(* IEC 61131-3 sources: Fosela-House-/control/free_evolution, 19 files *)

(* ---- GVL_Evolution.st ---- *)
(* ============================================================
   GVL_Evolution.st
   Variables globales del controlador principal (maestro Modbus).
   Sistema principal — Fosela House
   Arquitectura: BC monobloc genérica (sin HTR) + solar térmico
   ============================================================ *)

VAR_GLOBAL

    (* ---- Entradas analógicas locales (TT4-TT13) ---- *)
    TT4             : REAL;     (* D1 fondo — retorno agua técnica fría [°C] *)
    TT5             : REAL;     (* D2 cabeza — agua técnica caliente, salida a consumos [°C] *)
    TT6             : REAL;     (* Buffer D3 cabeza [°C] *)
    TT7             : REAL;     (* Buffer D3 fondo [°C] *)
    TT8             : REAL;     (* Ida primario BC [°C] *)
    TT9             : REAL;     (* Retorno primario BC [°C] *)
    TT11            : REAL;     (* Temperatura piscina [°C] *)
    TT12            : REAL;     (* Exterior [°C] *)
    TT13            : REAL;     (* Retorno fancoils [°C] *)

    (* ---- Entradas digitales ---- *)
    DI_Z1           : BOOL;     (* Termostato seguridad D1 activo *)
    DI_Z2           : BOOL;     (* Termostato seguridad D2 activo *)
    DI_INUND_FC     : BOOL;     (* Sensor inundación bandejas fancoils *)
    DI_BDC_FAULT    : BOOL;     (* Fallo BC (señal de la propia unidad) *)
    DI_IF_PISC      : BOOL;     (* Interruptor de flujo piscina *)

    (* ---- Salidas digitales ---- *)
    (* Distribución producción BC — dos V3V en cascada:
       V3V1: FALSE=Reservorio (D2 serpentines)  TRUE=→V3V2
       V3V2: FALSE=Buffer D3 fancoils           TRUE=HX_BC piscina *)
    DO_V3V1         : BOOL;     (* BC primario: FALSE=reservorio, TRUE=no-reservorio *)
    DO_V3V2         : BOOL;     (* no-reservorio: FALSE=fancoils (D3), TRUE=piscina (HX_BC) *)
    DO_VP_HX_SOLAR  : BOOL;     (* Válvula piscina lado HX solar *)
    DO_VP_HX_BC     : BOOL;     (* Válvula piscina lado HX aerotérmico *)
    DO_V3V_APT_01   : BOOL;     (* Aparto 1: FALSE=agua precalentada, TRUE=AFS red *)
    DO_V3V_APT_02   : BOOL;
    DO_V3V_APT_03   : BOOL;
    DO_V3V_APT_04   : BOOL;
    DO_P3           : BOOL;     (* Bomba fancoils arranque *)

    (* ---- Datos recibidos del controlador solar por Modbus ---- *)
    SM              : ST_SolarData;  (* Ver Types_Common.st *)

    (* ---- Modos y estados del sistema ---- *)
    bdc_mode        : E_BDC_Mode   := BDC_OFF;
    bdc_priority    : E_BDC_Priority := PRIO_ACS_CLIMATE_POOL;
    bc_mode_heat    : BOOL := TRUE;   (* TRUE=calefacción/ACS, FALSE=refrigeración *)

    (* ---- Ciclo de pasteurización ---- *)
    hyg_phase      : E_Hygienization_Phase := HYG_IDLE;
    hyg_request    : BOOL := FALSE;
    hyg_apt_idx    : UINT := 1;

    (* ---- Alarmas ---- *)
    alarms          : ST_SystemAlarms;

    (* ---- Setpoints enviados al controlador solar vía Modbus ---- *)
    P10_SolarDeltaTTarget           : UINT := 80;    (* 8.0 K ×10 *)
    P16_MinTempForPoolSolarHeating  : UINT := 750;   (* 75.0°C ×10 *)
    P17_SolarOverheatShutterClose   : UINT := 0;
    P19_SolarMode                   : UINT := 0;
    pool_demand_ext                 : UINT := 0;

END_VAR

(* ---- GVL_HMI_Params.st ---- *)
(* ============================================================
   GVL_HMI_Params.st
   Parámetros editables del HMI con sus rangos y valores por defecto.
   FUENTE ÚNICA DE VERDAD para todos los setpoints del sistema.
   Cualquier modificación desde el panel actualiza estas variables;
   la lógica de control las lee desde aquí.
   ============================================================ *)

VAR_GLOBAL RETAIN  (* RETAIN: sobreviven a un corte de alimentación *)

    (* ---- SOLAR ------------------------------------------ *)
    HMI_SP_DT_solar     : REAL := 8.0;   (* ΔT objetivo P1  [3.0 – 15.0 K]   paso 0.5 *)
    HMI_SP_TT3_pool     : REAL := 75.0;  (* TT3 → piscina   [60.0 – 90.0 °C] paso 1.0 *)
    HMI_modo_solar      : UINT := 0;     (* 0=AUTO 1=ACS 2=PISC 3=OFF *)

    (* ---- ACS -------------------------------------------- *)
    HMI_SP_TT5          : REAL := 65.0;  (* Setpoint D2 cab  [50.0 – 80.0 °C] paso 0.5 *)
    HMI_HS_TT5          : REAL := 3.0;   (* Histéresis TT5   [1.0 – 5.0 K]   paso 0.5 *)
    HMI_SP_TT4_start    : REAL := 50.0;  (* Umbral arrq BDC  [40.0 – 60.0 °C] paso 0.5 *)

    (* ---- CLIMATIZACIÓN ----------------------------------- *)
    HMI_SP_heat         : REAL := 45.0;  (* Setpoint calefac [35.0 – 60.0 °C] paso 0.5 *)
    HMI_SP_cool         : REAL := 9.0;   (* Setpoint refrig  [5.0 – 15.0 °C]  paso 0.5 *)
    HMI_HS_heat         : REAL := 2.0;   (* Histéresis calef [1.0 – 5.0 K]   paso 0.5 *)
    HMI_HS_cool         : REAL := 1.0;   (* Histéresis refrig[0.5 – 3.0 K]   paso 0.5 *)

    (* ---- PISCINA ---------------------------------------- *)
    HMI_SP_pool         : REAL := 27.0;  (* Setpoint piscina [20.0 – 35.0 °C] paso 0.5 *)
    HMI_HS_pool         : REAL := 1.0;   (* Histéresis pisc  [0.5 – 3.0 K]   paso 0.5 *)

    (* ---- PASTEURIZACIÓN --------------------------------- *)
    HMI_SP_past_target  : REAL := 70.0;  (* T objetivo past. [65.0 – 75.0 °C] paso 0.5 *)
    HMI_past_hold_min   : UINT := 60;    (* Tiempo manten.   [30 – 120 min]   paso 5   *)
    HMI_past_flush_min  : UINT := 30;    (* Tiempo purgado   [15 – 60 min]    paso 5   *)

    (* ---- APARTAMENTOS ----------------------------------- *)
    HMI_apt_mode_01     : UINT := 0;     (* 0=PRECALENTADA 1=AFS *)
    HMI_apt_mode_02     : UINT := 0;
    HMI_apt_mode_03     : UINT := 0;
    HMI_apt_mode_04     : UINT := 0;
    HMI_apt_mode_05     : UINT := 0;

    (* ---- CONFIGURACIÓN SISTEMA -------------------------- *)
    HMI_bdc_priority    : UINT := 0;     (* 0=ACS>CLIM>PISC  1=ACS>PISC>CLIM *)
    HMI_mb_slave_addr   : UINT := 1;     (* Dir. Modbus Smart [1 – 247] *)
    HMI_mb_baudrate     : UINT := 1;     (* 0=9600 1=19200 2=38400 *)

    (* ---- PIN DE ACCESO ---------------------------------- *)
    HMI_pin_test        : UINT := 1234;  (* PIN acceso TEST  [0 – 9999] *)
    HMI_pin_cfg         : UINT := 9999;  (* PIN acceso CFG   [0 – 9999] *)

END_VAR

(* ---- Variables de estado HMI (no RETAIN) ---- *)
VAR_GLOBAL

    (* Solicitudes de acción desde panel *)
    HMI_req_past_manual : BOOL := FALSE; (* Pulso: lanzar pasteurización *)
    HMI_req_alm_reset   : BOOL := FALSE; (* Pulso: reset alarmas *)
    HMI_req_factory_rst : BOOL := FALSE; (* Pulso: reset fábrica (CFG) *)

    (* Estado del HMI *)
    HMI_test_active     : BOOL := FALSE; (* Modo test activo *)
    HMI_cfg_active      : BOOL := FALSE; (* Modo config activo *)
    HMI_pin_ok          : BOOL := FALSE; (* PIN validado en sesión *)

    (* Página actual visible *)
    HMI_current_page    : UINT := 0;     (* 0=MAIN 1=SOL 2=ACS … *)

END_VAR

(* ---- FB_ACS.st ---- *)
(* ============================================================
   FB_ACS.st  –  Control de producción de ACS
   BC monobloc genérica (sin HTR).
   La BC puede producir ACS de dos formas según el equipo:
     a) Modo ACS dedicado (BDC_ACS): produce agua caliente 55-65°C
        directamente al reservorio (D2 serpentines).
     b) Inversión de ciclo (ACS como calefacción): misma V3V1,
        igual lógica, la BC produce caliente al reservorio.
   En ambos casos la lógica PLC es idéntica: V3V1 hacia reservorio
   y la BC en el modo que proceda.
   ============================================================ *)
FUNCTION_BLOCK FB_ACS
VAR_INPUT
    TT4             : REAL;  (* D1 fondo — agua técnica fría *)
    TT5             : REAL;  (* D2 cabeza — agua técnica caliente *)
    bdc_available   : BOOL;  (* BC autorizada por árbitro *)
    hyg_active      : BOOL;  (* Ciclo de higienización activo *)
    enabled         : BOOL := TRUE;
END_VAR
VAR_OUTPUT
    cmd_V3V1_reservorio : BOOL;  (* TRUE = BC primario → reservorio (D2) *)
    demand_BDC          : BOOL;  (* Solicitud al árbitro *)
    acs_satisfied       : BOOL;  (* Reservorio en setpoint *)
END_VAR
VAR
    ctrl_TT5    : FB_Hysteresis;
    ctrl_TT4    : FB_Hysteresis;
END_VAR

(* ACS satisfecho cuando TT5 (D2 cabeza) supera la consigna *)
ctrl_TT5(
    measured   := TT5,
    setpoint   := P30_ACSStorageSetPoint,
    hysteresis := P31_ACSStorageHysteresis,
    mode_heat  := TRUE,
    enabled    := enabled
);
acs_satisfied := NOT ctrl_TT5.output;

(* Demanda BC: cuando TT4 (fondo D1) cae bajo el umbral de arranque *)
ctrl_TT4(
    measured   := TT4,
    setpoint   := P32_ACSBDCStartTemp,
    hysteresis := P33_ACSBDCStartHyst,
    mode_heat  := TRUE,
    enabled    := enabled AND NOT acs_satisfied
);
demand_BDC := ctrl_TT4.output OR hyg_active;

(* V3V1: BC primario hacia reservorio cuando está autorizado *)
cmd_V3V1_reservorio := bdc_available AND (demand_BDC OR hyg_active);

END_FUNCTION_BLOCK

(* ---- FB_Alarms.st ---- *)
(* ============================================================
   FB_Alarms.st  –  Gestión centralizada de alarmas del sistema
   ============================================================ *)
FUNCTION_BLOCK FB_Alarms
VAR_INPUT
    TT1             : REAL;
    TT2             : REAL;
    TT5             : REAL;
    TT11            : REAL;
    comm_solar_ok   : BOOL;
    flow_pisc_ok    : BOOL;
    vp_any_open     : BOOL;
    inundacion      : BOOL;
    bdc_fault       : BOOL;
    reset_cmd       : BOOL;
    enabled         : BOOL := TRUE;
END_VAR
VAR_OUTPUT
    alarms          : ST_SystemAlarms;
    alarm_count     : UINT;
END_VAR
VAR
    alm_TT1         : FB_Alarm;
    alm_TT2         : FB_Alarm;
    alm_comm        : FB_Alarm;
    alm_TT5_low     : FB_Alarm;
    alm_TT5_high    : FB_Alarm;
    alm_pisc_flow   : FB_Alarm;
    alm_pisc_temp   : FB_Alarm;
    alm_inund       : FB_Alarm;
    alm_bdc         : FB_Alarm;
END_VAR

alm_TT1(condition := TT1 > P04_CollectorMaxOperTemp,
         reset_cmd := reset_cmd, filter_time := K_ALM_FILTER, latch := FALSE, enabled := enabled);
alm_TT2(condition := TT2 > (P00_AccumulatorMaxTemp - 7.0),
         reset_cmd := reset_cmd, filter_time := K_ALM_FILTER, latch := FALSE, enabled := enabled);
alm_comm(condition := NOT comm_solar_ok,
         reset_cmd := reset_cmd, filter_time := P93_ModbusTimeout, latch := TRUE, enabled := enabled);
alm_TT5_low(condition := TT5 < 40.0,
         reset_cmd := reset_cmd, filter_time := T#120M, latch := TRUE, enabled := enabled);
alm_TT5_high(condition := TT5 > (P00_AccumulatorMaxTemp - 5.0),
         reset_cmd := reset_cmd, filter_time := K_ALM_FILTER, latch := FALSE, enabled := enabled);
alm_pisc_flow(condition := NOT flow_pisc_ok AND vp_any_open,
         reset_cmd := reset_cmd, filter_time := T#30S, latch := TRUE, enabled := enabled);
alm_pisc_temp(condition := TT11 > P62_PoolMaxTemp,
         reset_cmd := reset_cmd, filter_time := K_ALM_FILTER, latch := FALSE, enabled := enabled);
alm_inund(condition := inundacion,
         reset_cmd := reset_cmd, filter_time := T#5S, latch := TRUE, enabled := enabled);
alm_bdc(condition := bdc_fault,
         reset_cmd := reset_cmd, filter_time := T#5S, latch := TRUE, enabled := enabled);

alarms.ALM_TT1_HIGH      := alm_TT1.active;
alarms.ALM_TT2_HIGH      := alm_TT2.active;
alarms.ALM_COMM_SOLAR    := alm_comm.active;
alarms.ALM_TT5_LOW       := alm_TT5_low.active;
alarms.ALM_TT5_HIGH      := alm_TT5_high.active;
alarms.ALM_PISC_FLUJO    := alm_pisc_flow.active;
alarms.ALM_PISC_T_HIGH   := alm_pisc_temp.active;
alarms.ALM_INUNDACION    := alm_inund.active;
alarms.ALM_BDC_FAULT     := alm_bdc.active;
alarms.CUALQUIER_ALARMA  :=
    alm_TT1.active OR alm_TT2.active OR alm_comm.active OR
    alm_TT5_low.active OR alm_TT5_high.active OR alm_pisc_flow.active OR
    alm_pisc_temp.active OR alm_inund.active OR alm_bdc.active;

alarm_count := 0;
IF alarms.ALM_TT1_HIGH    THEN alarm_count := alarm_count + 1; END_IF
IF alarms.ALM_TT2_HIGH    THEN alarm_count := alarm_count + 1; END_IF
IF alarms.ALM_COMM_SOLAR  THEN alarm_count := alarm_count + 1; END_IF
IF alarms.ALM_TT5_LOW     THEN alarm_count := alarm_count + 1; END_IF
IF alarms.ALM_TT5_HIGH    THEN alarm_count := alarm_count + 1; END_IF
IF alarms.ALM_PISC_FLUJO  THEN alarm_count := alarm_count + 1; END_IF
IF alarms.ALM_PISC_T_HIGH THEN alarm_count := alarm_count + 1; END_IF
IF alarms.ALM_INUNDACION  THEN alarm_count := alarm_count + 1; END_IF
IF alarms.ALM_BDC_FAULT   THEN alarm_count := alarm_count + 1; END_IF

END_FUNCTION_BLOCK

(* ---- FB_Apartments.st ---- *)
(* ============================================================
   FB_Apartments.st  –  Gestión V3V_APT por apartamento
   Modo por defecto: precalentada.
   Conmuta a AFS en mantenimiento, vacancia o higienización.
   ============================================================ *)
FUNCTION_BLOCK FB_Apartments
VAR_INPUT
    hyg_active          : BOOL;  (* Higienización activa → forzar precalentada *)
    maintenance_mode    : BOOL;  (* Mantenimiento central → AFS *)
    enabled             : BOOL := TRUE;
END_VAR
VAR_OUTPUT
    (* FALSE = precalentada (energiza), TRUE = AFS (desenergiza) *)
    cmd_APT_01 : BOOL;
    cmd_APT_02 : BOOL;
    cmd_APT_03 : BOOL;
    cmd_APT_04 : BOOL;
    cmd_APT_05 : BOOL;
END_VAR

(* Durante higienización: forzar precalentada en todos *)
IF hyg_active THEN
    cmd_APT_01 := FALSE;
    cmd_APT_02 := FALSE;
    cmd_APT_03 := FALSE;
    cmd_APT_04 := FALSE;
    cmd_APT_05 := FALSE;
ELSIF maintenance_mode THEN
    (* Mantenimiento central: todos a AFS *)
    cmd_APT_01 := TRUE;
    cmd_APT_02 := TRUE;
    cmd_APT_03 := TRUE;
    cmd_APT_04 := TRUE;
    cmd_APT_05 := TRUE;
ELSE
    (* Modo individual según ip_AptMode_XX *)
    cmd_APT_01 := (P40_AptMode_01 = UINT#1);
    cmd_APT_02 := (P41_AptMode_02 = UINT#1);
    cmd_APT_03 := (P42_AptMode_03 = UINT#1);
    cmd_APT_04 := (P43_AptMode_04 = UINT#1);
    cmd_APT_05 := (P44_AptMode_05 = UINT#1);
END_IF

END_FUNCTION_BLOCK

(* ---- FB_BDC_Arbiter.st ---- *)
(* ============================================================
   FB_BDC_Arbiter.st  –  Árbitro de prioridades del primario BDC
   Asigna el primario BDC a un único subsistema según P80_BDCPriority.
   Prioridad 0: ACS > Climatización > Piscina
   Prioridad 1: ACS > Piscina > Climatización
   ============================================================ *)
FUNCTION_BLOCK FB_BDC_Arbiter
VAR_INPUT
    demand_DHW      : BOOL;
    demand_climate  : BOOL;
    demand_pool     : BOOL;
    enabled         : BOOL := TRUE;
END_VAR
VAR_OUTPUT
    grant_DHW       : BOOL;
    grant_climate   : BOOL;
    grant_pool      : BOOL;
    active_mode     : E_BDC_Mode;
END_VAR

grant_DHW     := FALSE;
grant_climate := FALSE;
grant_pool    := FALSE;
active_mode   := BDC_OFF;

IF NOT enabled THEN RETURN; END_IF

IF demand_DHW THEN
    grant_DHW   := TRUE;
    active_mode := BDC_DHW;

ELSIF P80_BDCPriority = UINT#0 THEN
    (* ACS > Climatización > Piscina *)
    IF demand_climate THEN
        grant_climate := TRUE;
        active_mode   := BDC_CLIMATE;
    ELSIF demand_pool THEN
        grant_pool  := TRUE;
        active_mode := BDC_POOL;
    END_IF

ELSE
    (* ACS > Piscina > Climatización *)
    IF demand_pool THEN
        grant_pool  := TRUE;
        active_mode := BDC_POOL;
    ELSIF demand_climate THEN
        grant_climate := TRUE;
        active_mode   := BDC_CLIMATE;
    END_IF
END_IF

END_FUNCTION_BLOCK

(* ---- FB_Climate.st ---- *)
(* ============================================================
   FB_Climate.st  –  Control climatización fancoils
   Gestiona V3V2 (→D3), P3. Doble modo calor/frío.
   ============================================================ *)
FUNCTION_BLOCK FB_Climate
VAR_INPUT
    TT6             : REAL;  (* D3 cabeza *)
    TT7             : REAL;  (* D3 fondo *)
    bdc_available   : BOOL;
    mode_heat       : BOOL;  (* TRUE=calefacción FALSE=refrigeración *)
    enabled         : BOOL := TRUE;
END_VAR
VAR_OUTPUT
    cmd_V3V2_D3     : BOOL;  (* TRUE = primario BDC → D3 *)
    cmd_P3          : BOOL;  (* Bomba fancoils *)
    demand_BDC      : BOOL;
    climate_satisfied: BOOL;
END_VAR
VAR
    ctrl_heat : FB_Hysteresis;
    ctrl_cool : FB_Hysteresis;
    pump_P3   : FB_Pump;
END_VAR

IF mode_heat THEN
    ctrl_heat(
        measured   := TT6,
        setpoint   := P50_HeatingSetPoint,
        hysteresis := P51_HeatingHysteresis,
        mode_heat  := TRUE,
        enabled    := enabled
    );
    demand_BDC       := ctrl_heat.output;
    climate_satisfied := NOT ctrl_heat.output;
ELSE
    ctrl_cool(
        measured   := TT7,
        setpoint   := P52_CoolingSetPoint,
        hysteresis := P53_CoolingHysteresis,
        mode_heat  := FALSE,
        enabled    := enabled
    );
    demand_BDC       := ctrl_cool.output;
    climate_satisfied := NOT ctrl_cool.output;
END_IF

cmd_V3V2_D3 := bdc_available AND demand_BDC;

pump_P3(
    cmd_run     := cmd_V3V2_D3,
    min_on_time := T#60S,
    min_off_time:= T#30S,
    enabled     := enabled
);
cmd_P3 := pump_P3.DO_pump;

END_FUNCTION_BLOCK

(* ---- FB_ClimateReversible.st ---- *)
(* ============================================================
   FB_ClimateReversible.st
   Climatización reversible con buffer de inercia de 150 L como
   aguja hidráulica de 4 bocas.

   ARQUITECTURA:
   - Invierno (BC en calor): el primario del buffer se alimenta del
     TÁNDEM (D2). La bomba P1 (rama de invierno) circula el agua del
     tándem por el buffer. Así la SOLAR contribuye a calefacción.
   - Verano (BC en frío): el primario del buffer se alimenta de la BC
     en frío vía la V3V estacional. P1 parada (empuja la BC).
   - P2 (secundario) mueve el agua del buffer a los fancoils SIEMPRE.

   Conmutación de fuente con 4 válvulas de zona de 2 vías, por parejas
   de estación (lo fija el dibujo del esquema de principio):
     VZ1 = verano-impulsión   VZ2 = verano-retorno
     VZ3 = invierno-impulsión VZ4 = invierno-retorno

   ENCLAVAMIENTO: las válvulas deben estar en posición ANTES de que
   arranque P1 o cambie el modo de la BC. Se respeta tiempo de maniobra
   + retardo de seguridad.

   NADA HARDCODED: tiempos y consignas en GVL_Params.
   ============================================================ *)

FUNCTION_BLOCK FB_ClimateReversible

VAR_INPUT
    eBC_Mode        : E_BDC_Mode;   (* Modo actual de la BC: HEAT / COOL / OFF *)
    bClimateDemand  : BOOL;         (* Hay demanda de clima (termostatos zona) *)
    rTT_buffer      : REAL;         (* Temperatura buffer clima [°C] *)
    bEnable         : BOOL := TRUE;
END_VAR

VAR_OUTPUT
    bVZ1_open       : BOOL;     (* verano-impulsión *)
    bVZ2_open       : BOOL;     (* verano-retorno *)
    bVZ3_open       : BOOL;     (* invierno-impulsión *)
    bVZ4_open       : BOOL;     (* invierno-retorno *)
    bP1_run         : BOOL;     (* circuladora primario clima (invierno) *)
    bP2_run         : BOOL;     (* circuladora secundario → fancoils *)
    bV3V_Seasonal_B : BOOL;     (* V3V estacional: FALSE=D2(calor) / TRUE=buffer(frío) *)
    eSeason         : E_Season;
    bInterlockOK    : BOOL;     (* Válvulas en posición, seguro para arrancar *)
END_VAR

VAR
    eSeasonTarget   : E_Season;
    timer_interlock : TON;
    VZ1, VZ2, VZ3, VZ4 : FB_Valve2Way;
    P1, P2          : FB_Pump;
END_VAR

(* ---------- Determinar estación objetivo según modo BC ---------- *)
IF eBC_Mode = E_BDC_Mode.COOL THEN
    eSeasonTarget := E_Season.SUMMER;
ELSE
    eSeasonTarget := E_Season.WINTER; (* HEAT y OFF → configuración de invierno *)
END_IF

(* ---------- Mando de válvulas de zona por parejas de estación ---------- *)
(* Verano: VZ1+VZ2 abiertas, VZ3+VZ4 cerradas. Invierno: al revés. *)
VZ1(cmd_open := (eSeasonTarget = E_Season.SUMMER) AND bEnable,
    travel_time := GVL_Params.P64_PoolValveTravelTime);
VZ2(cmd_open := (eSeasonTarget = E_Season.SUMMER) AND bEnable,
    travel_time := GVL_Params.P64_PoolValveTravelTime);
VZ3(cmd_open := (eSeasonTarget = E_Season.WINTER) AND bEnable,
    travel_time := GVL_Params.P64_PoolValveTravelTime);
VZ4(cmd_open := (eSeasonTarget = E_Season.WINTER) AND bEnable,
    travel_time := GVL_Params.P64_PoolValveTravelTime);

bVZ1_open := VZ1.is_open;
bVZ2_open := VZ2.is_open;
bVZ3_open := VZ3.is_open;
bVZ4_open := VZ4.is_open;

(* ---------- Enclavamiento: confirmar pareja correcta en posición ---------- *)
IF eSeasonTarget = E_Season.SUMMER THEN
    bInterlockOK := VZ1.is_open AND VZ2.is_open
                    AND NOT VZ3.in_transit AND NOT VZ4.in_transit;
ELSE
    bInterlockOK := VZ3.is_open AND VZ4.is_open
                    AND NOT VZ1.in_transit AND NOT VZ2.in_transit;
END_IF

(* Retardo de seguridad tras alcanzar posición, antes de habilitar bombas *)
timer_interlock(IN := bInterlockOK, PT := GVL_Params.P55_SeasonInterlockDelay);

(* ---------- Estación confirmada solo cuando el enclavamiento es estable ---------- *)
IF timer_interlock.Q THEN
    eSeason := eSeasonTarget;
END_IF

(* ---------- V3V estacional: posición coordinada ---------- *)
(* FALSE = a D2 (carga tándem, invierno) ; TRUE = a buffer frío (verano) *)
bV3V_Seasonal_B := (eSeason = E_Season.SUMMER);

(* ---------- Bombas ---------- *)
(* P1 (primario clima) SOLO en invierno y con enclavamiento OK *)
P1(cmd_run := (eSeason = E_Season.WINTER) AND bClimateDemand AND timer_interlock.Q,
   min_on_time := GVL_Params.P14_SolarPumpMinOnTime,
   min_off_time := GVL_Params.P15_SolarPumpMinOffTime,
   enabled := bEnable);
bP1_run := P1.running;

(* P2 (secundario → fancoils) siempre que haya demanda y enclavamiento OK *)
P2(cmd_run := bClimateDemand AND timer_interlock.Q,
   enabled := bEnable);
bP2_run := P2.running;

(* ---- FB_DHW.st ---- *)
(* ============================================================
   FB_DHW.st  –  Control de producción de ACS
   BC monobloc genérica (sin HTR).
   La BC puede producir ACS de dos formas según el equipo:
     a) Modo ACS dedicado (BDC_DHW): produce agua caliente 55-65°C
        directamente al reservorio (D2 serpentines).
     b) Inversión de ciclo (ACS como calefacción): misma V3V1,
        igual lógica, la BC produce caliente al reservorio.
   En ambos casos la lógica PLC es idéntica: V3V1 hacia reservorio
   y la BC en el modo que proceda.
   ============================================================ *)
FUNCTION_BLOCK FB_DHW
VAR_INPUT
    TT4             : REAL;  (* D1 fondo — agua técnica fría *)
    TT5             : REAL;  (* D2 cabeza — agua técnica caliente *)
    bdc_available   : BOOL;  (* BC autorizada por árbitro *)
    hyg_active      : BOOL;  (* Ciclo de higienización activo *)
    enabled         : BOOL := TRUE;
END_VAR
VAR_OUTPUT
    cmd_V3V1_reservorio : BOOL;  (* TRUE = BC primario → reservorio (D2) *)
    demand_BDC          : BOOL;  (* Solicitud al árbitro *)
    acs_satisfied       : BOOL;  (* Reservorio en setpoint *)
END_VAR
VAR
    ctrl_TT5    : FB_Hysteresis;
    ctrl_TT4    : FB_Hysteresis;
END_VAR

(* ACS satisfecho cuando TT5 (D2 cabeza) supera la consigna *)
ctrl_TT5(
    measured   := TT5,
    setpoint   := P30_DHWStorageSetPoint,
    hysteresis := P31_DHWStorageHysteresis,
    mode_heat  := TRUE,
    enabled    := enabled
);
acs_satisfied := NOT ctrl_TT5.output;

(* Demanda BC: cuando TT4 (fondo D1) cae bajo el umbral de arranque *)
ctrl_TT4(
    measured   := TT4,
    setpoint   := P32_DHWBDCStartTemp,
    hysteresis := P33_DHWBDCStartHyst,
    mode_heat  := TRUE,
    enabled    := enabled AND NOT acs_satisfied
);
demand_BDC := ctrl_TT4.output OR hyg_active;

(* V3V1: BC primario hacia reservorio cuando está autorizado *)
cmd_V3V1_reservorio := bdc_available AND (demand_BDC OR hyg_active);

END_FUNCTION_BLOCK

(* ---- FB_DHW_Station.st ---- *)
(* ============================================================
   FB_DHW_Station.st
   Estación de producción de ACS al paso (agua fresca).
   Intercambiador de placas HX-ACS + circuladora P-ACS + caudalímetro
   YF-B6 + lazo PI sobre temperatura de salida de placa.

   NADA HARDCODED: todos los umbrales en GVL_Params.

   Lazo de control: PI (no PID) sobre TT_DHW_out → velocidad P-ACS.
   Detección de demanda por caudalímetro (anticipación).
   Parada suave (cooldown) para evacuar calor residual.
   Corte térmico bimetálico NC = seguro hardware independiente;
   aquí solo se LEE su estado para alarma y parada lógica.

   Estados: IDLE, ANTICIPATION, ACTIVE, COOLDOWN, PREHEATING,
            ALARM, INHIBITED
   ============================================================ *)

FUNCTION_BLOCK FB_DHW_Station

VAR_INPUT
    rFlowRate       : REAL;     (* Caudal secundario [L/min], calculado del HSC *)
    rTT_DHW_out     : REAL;     (* Temperatura salida placa (sonda rápida) [°C] *)
    rTT_DHW_ret     : REAL;     (* Temperatura retorno primario [°C] (diagnóstico) *)
    rTT5_Reservoir  : REAL;     (* Temperatura tapa D2 (reservorio) [°C] *)
    bThermalCutout  : BOOL;     (* Corte térmico NC: TRUE=normal, FALSE=disparado *)
    bEnable         : BOOL := TRUE; (* Habilitación desde árbitro BDC *)
    bPreheatRequest : BOOL := FALSE;(* Solicitud ciclo precalentamiento apartamentos *)
    dt_seconds      : REAL := 1.0;  (* Periodo de tarea [s] *)
END_VAR

VAR_OUTPUT
    rPACS_Speed     : REAL;     (* Consigna velocidad P-ACS [0..100 %] → TR0+buck *)
    eState          : E_DHW_Station_State;
    bAlarmCutout    : BOOL;     (* Corte térmico disparado *)
    bAlarmResLow    : BOOL;     (* Reservorio por debajo de mínimo crítico *)
    bAlarmOverTemp  : BOOL;     (* Sobretemperatura salida ACS *)
    bWarnResLow     : BOOL;     (* Reservorio bajo (aviso, no crítico) *)
END_VAR

VAR
    PI_DHW          : FB_PI_Controller;
    timer_cooldown  : TON;
    bFlowPresent    : BOOL;
END_VAR

(* ---------- Detección de presencia de flujo ---------- *)
bFlowPresent := rFlowRate >= GVL_Params.P37_DHWFlowDetectMin;

(* ---------- Vigilancia del reservorio ---------- *)
bWarnResLow  := rTT5_Reservoir < GVL_Params.P32_DHWReservoirMinForACS;
bAlarmResLow := rTT5_Reservoir < GVL_Params.P33_DHWReservoirAlarmLow;

(* ---------- Protecciones que fuerzan ALARM ---------- *)
bAlarmCutout   := NOT bThermalCutout;  (* contacto NC abierto = disparo *)
bAlarmOverTemp := rTT_DHW_out > GVL_Params.P39_DHWMaxOutputAlarm;

(* ============================================================
   MÁQUINA DE ESTADOS
   ============================================================ *)
IF bAlarmCutout OR bAlarmOverTemp OR bAlarmResLow THEN
    eState := E_DHW_Station_State.ALARM;
ELSIF NOT bEnable THEN
    eState := E_DHW_Station_State.INHIBITED;
END_IF

CASE eState OF

    E_DHW_Station_State.IDLE:
        rPACS_Speed := 0.0;
        PI_DHW.reset := TRUE;
        IF bFlowPresent THEN
            eState := E_DHW_Station_State.ANTICIPATION;
        ELSIF bPreheatRequest THEN
            eState := E_DHW_Station_State.PREHEATING;
        END_IF

    E_DHW_Station_State.ANTICIPATION:
        (* Arranque inmediato al primer pulso, antes de que caiga la T *)
        PI_DHW.reset := FALSE;
        rPACS_Speed := GVL_Params.P13_SolarPumpMinSpeed; (* arranque suave *)
        eState := E_DHW_Station_State.ACTIVE;

    E_DHW_Station_State.ACTIVE:
        (* Lazo PI: mantener TT_DHW_out en consigna de placa *)
        PI_DHW(measured := rTT_DHW_out,
               setpoint := GVL_Params.P34_DHWPlateOutputSetpoint,
               Kp := GVL_Params.P22_DHWPI_Kp,
               Ki := GVL_Params.P23_DHWPI_Ki,
               out_min := GVL_Params.P13_SolarPumpMinSpeed,
               out_max := 100.0,
               dt_seconds := dt_seconds,
               enabled := TRUE);
        rPACS_Speed := PI_DHW.output;
        IF NOT bFlowPresent THEN
            timer_cooldown(IN := FALSE);
            eState := E_DHW_Station_State.COOLDOWN;
        END_IF

    E_DHW_Station_State.COOLDOWN:
        (* Mantener bomba un tiempo para evacuar calor residual de la placa *)
        rPACS_Speed := GVL_Params.P13_SolarPumpMinSpeed;
        timer_cooldown(IN := TRUE, PT := GVL_Params.P38_DHWPumpCooldown);
        IF bFlowPresent THEN
            timer_cooldown(IN := FALSE);
            eState := E_DHW_Station_State.ACTIVE;
        ELSIF timer_cooldown.Q THEN
            timer_cooldown(IN := FALSE);
            eState := E_DHW_Station_State.IDLE;
        END_IF

    E_DHW_Station_State.PREHEATING:
        (* Precalentamiento de termos de apartamentos: la apertura
           secuencial de V3V_APT la gestiona FB_Preheating; aquí solo
           se asegura caudal por la placa. *)
        rPACS_Speed := 60.0;  (* caudal medio fijo durante precalentamiento *)
        IF NOT bPreheatRequest THEN
            eState := E_DHW_Station_State.COOLDOWN;
        ELSIF bFlowPresent THEN
            eState := E_DHW_Station_State.ACTIVE; (* demanda real tiene prioridad *)
        END_IF

    E_DHW_Station_State.ALARM:
        rPACS_Speed := 0.0;        (* parada lógica; el hardware ya cortó *)
        PI_DHW.reset := TRUE;
        IF NOT bAlarmCutout AND NOT bAlarmOverTemp AND NOT bAlarmResLow THEN
            eState := E_DHW_Station_State.IDLE;  (* corte térmico es rearme manual:
                                                    bThermalCutout vuelve a TRUE solo
                                                    tras rearme físico *)
        END_IF

    E_DHW_Station_State.INHIBITED:
        rPACS_Speed := 0.0;
        PI_DHW.reset := TRUE;
        IF bEnable THEN
            eState := E_DHW_Station_State.IDLE;
        END_IF

END_CASE

(* ---- FB_HybridOptimizer.st ---- *)
(* ============================================================
   FB_HybridOptimizer.st
   Optimizador de fuente BC: Agua-Agua vs Aire-Agua

   PRINCIPIO MATEMÁTICO:
   ─────────────────────
   COP_WW_cal = η·(T_cond+273) / [T_cond − (T_pool − ΔT_ap)]
   COP_AW_cal = η·(T_cond+273) / [T_cond − T_air]

   COP_WW > COP_AW  ⟺  T_pool − ΔT_ap > T_air
                    ⟺  T_pool > T_air + ΔT_ap     [calefacción]

   COP_WW_frio = η·(T_evap+273) / [(T_pool + ΔT_ap) − T_evap]
   COP_AW_frio = η·(T_evap+273) / [T_air − T_evap]

   COP_WW > COP_AW  ⟺  T_pool + ΔT_ap < T_air
                    ⟺  T_pool < T_air − ΔT_ap     [refrigeración]

   El umbral óptimo de conmutación ES la temperatura de approach
   del intercambiador agua↔refrigerante. No es un parámetro
   heurístico: es la condición exacta de igualdad de COPs.

   Con histéresis para evitar cicleo en la zona de indiferencia.
   ============================================================ *)

FUNCTION_BLOCK FB_HybridOptimizer
VAR_INPUT
    T_pool          : REAL;     (* Temperatura piscina [°C] *)
    T_air           : REAL;     (* Temperatura exterior [°C] *)
    mode_heat       : BOOL;     (* TRUE=calefacción/ACS, FALSE=refrigeración *)
    pool_available  : BOOL;     (* Piscina operativa (T_pool > T_pool_min) *)
    enabled         : BOOL := TRUE;
END_VAR

VAR_OUTPUT
    use_WW          : BOOL;     (* TRUE = usar BC agua-agua *)
    use_AW          : BOOL;     (* TRUE = usar BC aire-agua *)
    COP_WW          : REAL;     (* COP calculado BC agua-agua *)
    COP_AW          : REAL;     (* COP calculado BC aire-agua *)
    COP_advantage   : REAL;     (* % ventaja de la fuente elegida vs la otra *)
    source_str      : STRING;   (* "WW" o "AW" para HMI *)
END_VAR

VAR
    (* Parámetros termodinámicos — configurables en puesta en marcha *)
    eta_carnot      : REAL := 0.50;   (* Eficiencia relativa al Carnot *)
    T_cond_cal      : REAL := 47.0;   (* °C condensación modo calefacción *)
    T_evap_ref      : REAL := 7.0;    (* °C evaporación modo refrigeración *)
    DT_approach     : REAL := 5.0;    (* K approach agua↔refrigerante *)
    histeresis      : REAL := 1.5;    (* K banda muerta para evitar cicleo *)

    (* Estado interno *)
    last_use_WW     : BOOL := FALSE;
    timer_min_run   : TON;
    MIN_RUN_TIME    : TIME := T#10M;  (* Tiempo mínimo en cada modo *)

    (* Variables de cálculo *)
    denom_WW        : REAL;
    denom_AW        : REAL;
    threshold       : REAL;
    T_cond_K        : REAL;
    T_evap_K        : REAL;
END_VAR

(* ── Protección denominadores ────────────────────────────── *)
T_cond_K := T_cond_cal + 273.15;
T_evap_K  := T_evap_ref + 273.15;

IF NOT enabled OR NOT pool_available THEN
    use_WW      := FALSE;
    use_AW      := TRUE;
    COP_WW      := 0.0;
    COP_AW      := 0.0;
    COP_advantage:= 0.0;
    source_str  := 'AW';
    RETURN;
END_IF

(* ── Calcular COPs reales ────────────────────────────────── *)
IF mode_heat THEN
    (* Calefacción: evap en piscina (WW) o en aire (AW), cond en edificio *)
    denom_WW := T_cond_cal - (T_pool - DT_approach);
    denom_AW := T_cond_cal - T_air;
    IF denom_WW < 3.0 THEN denom_WW := 3.0; END_IF
    IF denom_AW < 3.0 THEN denom_AW := 3.0; END_IF
    COP_WW := eta_carnot * T_cond_K / denom_WW;
    COP_AW := eta_carnot * T_cond_K / denom_AW;

    (* Umbral analítico: T_pool = T_air + DT_approach *)
    threshold := T_air + DT_approach;

ELSE
    (* Refrigeración: evap en edificio, cond en piscina (WW) o en aire (AW) *)
    denom_WW := (T_pool + DT_approach) - T_evap_ref;
    denom_AW := T_air - T_evap_ref;
    IF denom_WW < 3.0 THEN denom_WW := 3.0; END_IF
    IF denom_AW < 3.0 THEN denom_AW := 3.0; END_IF
    COP_WW := eta_carnot * T_evap_K / denom_WW;
    COP_AW := eta_carnot * T_evap_K / denom_AW;

    (* Umbral analítico: T_pool = T_air - DT_approach *)
    threshold := T_air - DT_approach;
END_IF

(* ── Decisión con histéresis ─────────────────────────────── *)
(* Timer mínimo: no conmutar si llevamos menos de MIN_RUN_TIME en el modo actual *)
timer_min_run(IN := TRUE, PT := MIN_RUN_TIME);

IF timer_min_run.Q THEN
    (* Permitido conmutar: aplicar histéresis *)
    IF mode_heat THEN
        IF T_pool > threshold + histeresis THEN
            last_use_WW := TRUE;   timer_min_run(IN:=FALSE);
        ELSIF T_pool < threshold - histeresis THEN
            last_use_WW := FALSE;  timer_min_run(IN:=FALSE);
        END_IF
        (* Entre ±histeresis: mantener el modo anterior *)
    ELSE
        (* Refrigeración: WW mejor cuando piscina MÁS FRÍA que el umbral *)
        IF T_pool < threshold - histeresis THEN
            last_use_WW := TRUE;   timer_min_run(IN:=FALSE);
        ELSIF T_pool > threshold + histeresis THEN
            last_use_WW := FALSE;  timer_min_run(IN:=FALSE);
        END_IF
    END_IF
END_IF

(* ── Salidas ─────────────────────────────────────────────── *)
use_WW := last_use_WW;
use_AW := NOT last_use_WW;

IF use_WW THEN
    source_str    := 'WW';
    IF COP_AW > 0.0 THEN
        COP_advantage := (COP_WW - COP_AW) / COP_AW * 100.0;
    END_IF
ELSE
    source_str    := 'AW';
    IF COP_WW > 0.0 THEN
        COP_advantage := (COP_AW - COP_WW) / COP_WW * 100.0;
    END_IF
END_IF

END_FUNCTION_BLOCK

(* ============================================================
   NOTA DE IMPLEMENTACIÓN PARA FREE STUDIO
   ─────────────────────────────────────────
   Entradas físicas necesarias:
     TT11 → T_pool (sonda NTC en piscina, ya existente)
     TT12 → T_air  (sonda NTC exterior, ya existente)

   Salidas digitales:
     DO_SEL_WW → Activa circuito agua-agua (abre V_WW, arranca P_circ_ww)
     DO_SEL_AW → Activa circuito aire-agua (selecciona modo AW en BC)

   Variables HMI a mapear:
     COP_WW, COP_AW, COP_advantage, source_str

   El bloque se llama en PLC_PRG_Evolution antes de FB_BDC_Arbiter.
   use_WW / use_AW condicionan qué circuito de fuente se activa
   antes de que el árbitro asigne el modo (cal/frio/ACS/piscina).
   ============================================================ *)

(* ---- FB_Hygienization.st ---- *)
(* ============================================================
   FB_Hygienization.st  –  Ciclo de higienización térmica
   Máquina de estados: IDLE → HEAT_D2 → HOLD_D2 → FLUSH → DONE
   ============================================================ *)
FUNCTION_BLOCK FB_Hygienization
VAR_INPUT
    TT5             : REAL;
    manual_request  : BOOL;
    enabled         : BOOL := TRUE;
END_VAR
VAR_OUTPUT
    phase           : E_Hygienization_Phase;
    active          : BOOL;
    apt_idx         : UINT;   (* Apartamento actual en purgado 1-5 *)
    force_BDC_ACS   : BOOL;   (* Forzar BDC a modo ACS *)
    force_APT_prec  : BOOL;   (* Forzar V3V_APT a precalentada *)
END_VAR
VAR
    timer_hold      : TON;
    timer_flush     : TON;
    ctrl_hyg        : FB_Hysteresis;
    r_manual        : R_TRIG;
    scheduled_trigger: BOOL;  (* TODO: conectar al programador horario *)
END_VAR

r_manual(CLK := manual_request);

CASE phase OF

HYG_IDLE:
    active         := FALSE;
    force_BDC_ACS  := FALSE;
    force_APT_prec := FALSE;
    apt_idx        := 1;
    timer_hold(IN := FALSE, PT := P72_HygienizationHoldTime);
    timer_flush(IN := FALSE, PT := P73_HygienizationFlushTime);
    IF (r_manual.Q OR scheduled_trigger) AND enabled THEN
        phase := HYG_HEAT_D2;
    END_IF

HYG_HEAT_D2:
    active        := TRUE;
    force_BDC_ACS := TRUE;
    force_APT_prec:= TRUE;
    ctrl_hyg(
        measured   := TT5,
        setpoint   := P70_HygienizationTarget,
        hysteresis := P71_HygienizationHysteresis,
        mode_heat  := TRUE
    );
    IF NOT ctrl_hyg.output THEN
        phase := HYG_HOLD_D2;
    END_IF

HYG_HOLD_D2:
    active        := TRUE;
    force_BDC_ACS := TRUE;
    force_APT_prec:= TRUE;
    timer_hold(IN := TRUE, PT := P72_HygienizationHoldTime);
    IF timer_hold.Q THEN
        timer_hold(IN := FALSE, PT := P72_HygienizationHoldTime);
        phase   := HYG_FLUSH;
        apt_idx := 1;
    END_IF

HYG_FLUSH:
    active        := TRUE;
    force_BDC_ACS := TRUE;
    force_APT_prec:= TRUE;
    timer_flush(IN := TRUE, PT := P73_HygienizationFlushTime);
    IF timer_flush.Q THEN
        timer_flush(IN := FALSE, PT := P73_HygienizationFlushTime);
        IF apt_idx < 5 THEN
            apt_idx := apt_idx + 1;
        ELSE
            phase := HYG_DONE;
        END_IF
    END_IF

HYG_DONE:
    active        := FALSE;
    force_BDC_ACS := FALSE;
    force_APT_prec:= FALSE;
    phase         := HYG_IDLE;

END_CASE

END_FUNCTION_BLOCK

(* ---- FB_PIN_Guard.st ---- *)
(* ============================================================
   FB_PIN_Guard.st
   Gestión de acceso con PIN a menús restringidos (TEST, CFG).
   - Muestra "PIN:" en display y permite introducir 4 dígitos.
   - Bloqueo automático tras 3 intentos fallidos (5 minutos).
   - Timeout de sesión: cierra acceso tras inactividad.
   ============================================================ *)

FUNCTION_BLOCK FB_PIN_Guard

VAR_INPUT
    pin_stored      : UINT;             (* PIN configurado *)
    pin_entered     : UINT;             (* PIN introducido por operador *)
    confirm         : BOOL;             (* Pulso ENTER: validar PIN *)
    cancel          : BOOL;             (* Pulso ESC: cancelar *)
    activity        : BOOL;             (* TRUE si hay actividad en panel *)
    session_timeout : TIME := T#5M;     (* Tiempo de inactividad → cierre sesión *)
    lockout_time    : TIME := T#5M;     (* Tiempo de bloqueo tras 3 fallos *)
END_VAR

VAR_OUTPUT
    access_granted  : BOOL := FALSE;    (* TRUE = acceso concedido *)
    locked_out      : BOOL := FALSE;    (* TRUE = bloqueado por intentos *)
    attempts_left   : UINT := 3;        (* Intentos restantes *)
    show_error      : BOOL := FALSE;    (* Mostrar "Err" en display *)
END_VAR

VAR
    failed_attempts : UINT := 0;
    timer_session   : TON;
    timer_lockout   : TON;
    timer_error_msg : TON;
    r_confirm       : R_TRIG;
    r_cancel        : R_TRIG;
END_VAR

(* --- Detección de flancos --- *)
r_confirm(CLK := confirm);
r_cancel(CLK := cancel);

(* --- Bloqueo por intentos fallidos --- *)
timer_lockout(IN := locked_out, PT := lockout_time);
IF timer_lockout.Q THEN
    locked_out      := FALSE;
    failed_attempts := 0;
    timer_lockout(IN := FALSE, PT := lockout_time);
END_IF

(* --- Timeout de sesión por inactividad --- *)
timer_session(IN := access_granted AND NOT activity, PT := session_timeout);
IF timer_session.Q THEN
    access_granted := FALSE;
    timer_session(IN := FALSE, PT := session_timeout);
END_IF

(* --- Validación PIN --- *)
IF r_confirm.Q AND NOT locked_out AND NOT access_granted THEN
    IF pin_entered = pin_stored THEN
        access_granted  := TRUE;
        failed_attempts := 0;
        show_error      := FALSE;
    ELSE
        failed_attempts := failed_attempts + 1;
        show_error      := TRUE;
        timer_error_msg(IN := FALSE, PT := T#2S);
        IF failed_attempts >= 3 THEN
            locked_out := TRUE;
        END_IF
    END_IF
END_IF

(* Ocultar mensaje de error tras 2 segundos *)
timer_error_msg(IN := show_error, PT := T#2S);
IF timer_error_msg.Q THEN
    show_error := FALSE;
    timer_error_msg(IN := FALSE, PT := T#2S);
END_IF

(* --- Cancelar / cerrar sesión --- *)
IF r_cancel.Q THEN
    access_granted := FALSE;
END_IF

attempts_left := 3 - failed_attempts;

END_FUNCTION_BLOCK

(* ---- FB_Pool.st ---- *)
(* ============================================================
   FB_Pool.st  –  Control calentamiento/disipación piscina
   Dos intercambiadores de titanio independientes:
     HX_SOLAR : excedente solar → piscina
     HX_BC    : producción BC (solo en modo calefacción) → piscina
   La depuradora (P_DEPUR, existente) circula el agua de piscina
   por el secundario de ambos HX simultáneamente.
   ============================================================ *)
FUNCTION_BLOCK FB_Pool
VAR_INPUT
    TT11            : REAL;  (* Temperatura piscina [°C] *)
    solar_available : BOOL;  (* Solar excedente autorizado vía V3V_SOL *)
    bdc_available   : BOOL;  (* BC autorizado por árbitro AND en modo calor *)
    flow_ok         : BOOL;  (* Interruptor de flujo piscina activo *)
    enabled         : BOOL := TRUE;
END_VAR
VAR_OUTPUT
    cmd_VP_HX_SOLAR : BOOL;  (* Abrir válvula HX solar → piscina *)
    cmd_VP_HX_BC    : BOOL;  (* Abrir válvula HX aerotérmico → piscina *)
    demand_solar    : BOOL;  (* Solicitud aporte solar *)
    demand_BDC      : BOOL;  (* Solicitud aporte BC *)
    pool_satisfied  : BOOL;
    alarm_max_temp  : BOOL;
END_VAR
VAR
    ctrl_pool   : FB_Hysteresis;
    alm_max     : FB_Alarm;
END_VAR

ctrl_pool(
    measured   := TT11,
    setpoint   := P60_PoolSetPoint,
    hysteresis := P61_PoolHysteresis,
    mode_heat  := TRUE,
    enabled    := enabled
);
pool_satisfied := NOT ctrl_pool.output;

demand_solar := ctrl_pool.output AND flow_ok AND enabled;
demand_BDC   := ctrl_pool.output AND flow_ok AND enabled;

cmd_VP_HX_SOLAR := solar_available AND demand_solar;
cmd_VP_HX_BC    := bdc_available   AND demand_BDC;

alm_max(
    condition   := TT11 > P62_PoolMaxTemp,
    filter_time := K_ALM_FILTER,
    latch       := FALSE,
    enabled     := enabled
);
alarm_max_temp := alm_max.active;

IF alarm_max_temp THEN
    cmd_VP_HX_SOLAR := FALSE;
    cmd_VP_HX_BC    := FALSE;
END_IF

END_FUNCTION_BLOCK

(* ---- FB_Preheating.st ---- *)
(* ============================================================
   FB_Preheating.st  –  Ciclo de higienización térmica
   Máquina de estados: IDLE → HEAT_D2 → HOLD_D2 → FLUSH → DONE
   ============================================================ *)
FUNCTION_BLOCK FB_Preheating
VAR_INPUT
    TT5             : REAL;
    manual_request  : BOOL;
    enabled         : BOOL := TRUE;
END_VAR
VAR_OUTPUT
    phase           : E_Preheating_Phase;
    active          : BOOL;
    apt_idx         : UINT;   (* Apartamento actual en purgado 1-5 *)
    force_BDC_ACS   : BOOL;   (* Forzar BDC a modo ACS *)
    force_APT_prec  : BOOL;   (* Forzar V3V_APT a precalentada *)
END_VAR
VAR
    timer_hold      : TON;
    timer_flush     : TON;
    ctrl_hyg        : FB_Hysteresis;
    r_manual        : R_TRIG;
    scheduled_trigger: BOOL;  (* TODO: conectar al programador horario *)
END_VAR

r_manual(CLK := manual_request);

CASE phase OF

PRE_IDLE:
    active         := FALSE;
    force_BDC_ACS  := FALSE;
    force_APT_prec := FALSE;
    apt_idx        := 1;
    timer_hold(IN := FALSE, PT := P72_PreheatingHoldTime);
    timer_flush(IN := FALSE, PT := P73_PreheatingFlushTime);
    IF (r_manual.Q OR scheduled_trigger) AND enabled THEN
        phase := PRE_HEAT;
    END_IF

PRE_HEAT:
    active        := TRUE;
    force_BDC_ACS := TRUE;
    force_APT_prec:= TRUE;
    ctrl_hyg(
        measured   := TT5,
        setpoint   := P70_PreheatingTarget,
        hysteresis := P71_PreheatingHysteresis,
        mode_heat  := TRUE
    );
    IF NOT ctrl_hyg.output THEN
        phase := PRE_HOLD;
    END_IF

PRE_HOLD:
    active        := TRUE;
    force_BDC_ACS := TRUE;
    force_APT_prec:= TRUE;
    timer_hold(IN := TRUE, PT := P72_PreheatingHoldTime);
    IF timer_hold.Q THEN
        timer_hold(IN := FALSE, PT := P72_PreheatingHoldTime);
        phase   := PRE_FLUSH;
        apt_idx := 1;
    END_IF

PRE_FLUSH:
    active        := TRUE;
    force_BDC_ACS := TRUE;
    force_APT_prec:= TRUE;
    timer_flush(IN := TRUE, PT := P73_PreheatingFlushTime);
    IF timer_flush.Q THEN
        timer_flush(IN := FALSE, PT := P73_PreheatingFlushTime);
        IF apt_idx < 5 THEN
            apt_idx := apt_idx + 1;
        ELSE
            phase := PRE_DONE;
        END_IF
    END_IF

PRE_DONE:
    active        := FALSE;
    force_BDC_ACS := FALSE;
    force_APT_prec:= FALSE;
    phase         := PRE_IDLE;

END_CASE

END_FUNCTION_BLOCK

(* ---- FB_Solar.st ---- *)
(* ============================================================
   FB_Solar.st
   Control del circuito solar primario (glicol) con:
   - MUESTREO A BAJO CAUDAL: arranque por intervalos en lugar de
     sonda de captador. La bomba P-SOL arranca al mínimo caudal
     periódicamente para "tomar muestra" de lo que baja del campo
     sin consumir apenas energía ni disipar calor del depósito.
   - Modulación PI sobre ΔT (ida-retorno) con la bomba en marcha.
   - DISIPACIÓN ENCADENADA: 1º desvío a piscina (HX-POOL-SOL) si
     admite calor (< P62_PoolMaxTemp); 2º cierre de persianas.

   NADA HARDCODED: umbrales en GVL_Params.

   Estados: SLEEP, SAMPLING, RUNNING, DISSIPATING, OVERHEAT
   ============================================================ *)

FUNCTION_BLOCK FB_Solar

VAR_INPUT
    rTT_glycol_in   : REAL;     (* Ida: glicol que baja del campo [°C] *)
    rTT_glycol_out  : REAL;     (* Retorno: glicol frío hacia el campo [°C] *)
    rTT_D1          : REAL;     (* Temperatura D1 (depósito solar) [°C] *)
    rTT_pool        : REAL;     (* Temperatura piscina [°C] *)
    bEnable         : BOOL := TRUE;
    dt_seconds      : REAL := 1.0;
END_VAR

VAR_OUTPUT
    rPSOL_Speed     : REAL;     (* Consigna velocidad P-SOL [0..100 %] *)
    bV3V_Dissip_Pool: BOOL;     (* TRUE = V3V de disipación desvía a HX-POOL-SOL *)
    bShutterClose   : BOOL;     (* TRUE = cerrar persianas (último recurso) *)
    eState          : E_Solar_State;
    rDeltaT         : REAL;     (* ΔT actual ida-retorno [K] (diagnóstico) *)
END_VAR

VAR
    PI_Solar        : FB_PI_Controller;
    timer_interval  : TON;      (* Espera entre muestreos *)
    timer_sample    : TON;      (* Duración de la ventana de muestreo *)
    bReservoirFull  : BOOL;
    bPoolCanTake    : BOOL;
    rDeltaT_sample  : REAL;     (* ΔT respecto al depósito en el muestreo *)
END_VAR

(* ---------- Cálculos auxiliares ---------- *)
rDeltaT        := rTT_glycol_in - rTT_glycol_out;
rDeltaT_sample := rTT_glycol_in - rTT_D1;
bReservoirFull := rTT_D1 >= GVL_Params.P00_AccumulatorMaxTemp;
bPoolCanTake   := rTT_pool < GVL_Params.P62_PoolMaxTemp;

IF NOT bEnable THEN
    eState := E_Solar_State.SLEEP;
END_IF

(* ============================================================
   MÁQUINA DE ESTADOS
   ============================================================ *)
CASE eState OF

    E_Solar_State.SLEEP:
        (* Bomba parada. Esperar intervalo y muestrear. *)
        rPSOL_Speed := 0.0;
        bV3V_Dissip_Pool := FALSE;
        bShutterClose := FALSE;
        PI_Solar.reset := TRUE;
        timer_interval(IN := bEnable, PT := GVL_Params.P56_SolarSampleInterval);
        IF timer_interval.Q THEN
            timer_interval(IN := FALSE);
            timer_sample(IN := FALSE);
            eState := E_Solar_State.SAMPLING;
        END_IF

    E_Solar_State.SAMPLING:
        (* Bomba a BAJO CAUDAL: mínimo consumo, mínima disipación.
           Esperar a que el glicol del campo llegue a la sonda de ida. *)
        rPSOL_Speed := GVL_Params.P13_SolarPumpMinSpeed;
        PI_Solar.reset := TRUE;
        timer_sample(IN := TRUE, PT := GVL_Params.P57_SolarSampleDuration);
        IF timer_sample.Q THEN
            timer_sample(IN := FALSE);
            IF rDeltaT_sample >= GVL_Params.P11_SolarDeltaTStart THEN
                IF bReservoirFull THEN
                    eState := E_Solar_State.DISSIPATING;
                ELSE
                    eState := E_Solar_State.RUNNING;
                END_IF
            ELSE
                eState := E_Solar_State.SLEEP;  (* no merece la pena *)
            END_IF
        END_IF

    E_Solar_State.RUNNING:
        (* Carga normal a D1. PI mantiene ΔT objetivo modulando caudal. *)
        bV3V_Dissip_Pool := FALSE;
        bShutterClose := FALSE;
        PI_Solar(measured := rDeltaT,
                 setpoint := GVL_Params.P10_SolarDeltaTTarget,
                 Kp := GVL_Params.P20_SolarPI_Kp,
                 Ki := GVL_Params.P21_SolarPI_Ki,
                 out_min := GVL_Params.P13_SolarPumpMinSpeed,
                 out_max := 100.0,
                 dt_seconds := dt_seconds,
                 enabled := TRUE);
        rPSOL_Speed := PI_Solar.output;
        IF rDeltaT_sample < GVL_Params.P12_SolarDeltaTStop THEN
            eState := E_Solar_State.SLEEP;       (* campo agotado *)
        ELSIF bReservoirFull THEN
            eState := E_Solar_State.DISSIPATING; (* reservorio lleno *)
        END_IF

    E_Solar_State.DISSIPATING:
        (* 1er escalón: desviar excedente a la piscina si admite calor. *)
        IF bPoolCanTake THEN
            bV3V_Dissip_Pool := TRUE;
            bShutterClose := FALSE;
            rPSOL_Speed := PI_Solar.output;      (* seguir circulando hacia piscina *)
            IF rPSOL_Speed < GVL_Params.P13_SolarPumpMinSpeed THEN
                rPSOL_Speed := GVL_Params.P13_SolarPumpMinSpeed;
            END_IF
            IF NOT bReservoirFull THEN
                eState := E_Solar_State.RUNNING; (* hay sitio otra vez en D1 *)
            END_IF
        ELSE
            eState := E_Solar_State.OVERHEAT;    (* piscina llena: no hay sumidero *)
        END_IF

    E_Solar_State.OVERHEAT:
        (* 2º escalón: cerrar persianas y rezar. Defensa pasiva. *)
        bShutterClose := TRUE;
        bV3V_Dissip_Pool := FALSE;
        rPSOL_Speed := 0.0;
        PI_Solar.reset := TRUE;
        (* Reapertura con histéresis cuando baje la radiación/temperatura *)
        IF rTT_glycol_in < (GVL_Params.P17_SolarOverheatShutterClose
                            - GVL_Params.P18_SolarOverheatShutterHyst) THEN
            eState := E_Solar_State.SLEEP;
        ELSIF bPoolCanTake AND NOT bReservoirFull THEN
            eState := E_Solar_State.RUNNING;
        END_IF

END_CASE

(* ---- FB_TestMode.st ---- *)
(* ============================================================
   FB_TestMode.st
   Forzado manual de salidas para puesta en marcha y diagnóstico.
   SOLO activo si HMI_test_active = TRUE (acceso con PIN).
   Cuando test_active = FALSE todas las salidas de test se ponen
   a FALSE y el control normal retoma el mando.

   USO:
     Llamar en PLC_PRG_Evolution ANTES de las lógicas normales.
     Si test_active=TRUE las salidas del sistema se sobreescriben
     con los valores de test al FINAL del ciclo (mayor prioridad).
   ============================================================ *)

FUNCTION_BLOCK FB_TestMode

VAR_INPUT
    test_active         : BOOL;         (* TRUE = modo test habilitado *)
END_VAR

(* Comandos de test (editables desde HMI) *)
VAR_INPUT
    tst_P1_on           : BOOL;
    tst_P2_on           : BOOL;
    tst_P3_on           : BOOL;
    tst_P4_on           : BOOL;
    tst_V3V1_B          : BOOL;         (* TRUE = posición B *)
    tst_V3V2_B          : BOOL;
    tst_V3V3_B          : BOOL;
    tst_V3VSOL_B        : BOOL;
    tst_VP_HX1_open     : BOOL;
    tst_VP_HX_BDC_open  : BOOL;
    tst_VP_HX_HTR_open  : BOOL;
    tst_EV_BYPASS_open  : BOOL;
    tst_APT01_AFS       : BOOL;
    tst_APT02_AFS       : BOOL;
    tst_APT03_AFS       : BOOL;
    tst_APT04_AFS       : BOOL;
    tst_APT05_AFS       : BOOL;
    tst_PERS_close      : BOOL;
    tst_P1_speed_pct    : REAL := 50.0; (* Velocidad P1 test [0-100%] *)
END_VAR

VAR_OUTPUT
    (* Estas salidas sobreescriben las del sistema si test_active=TRUE *)
    out_DO_V3V1         : BOOL;
    out_DO_V3V2         : BOOL;
    out_DO_V3V3         : BOOL;
    out_DO_V3VSOL       : BOOL;
    out_DO_VP_HX1       : BOOL;
    out_DO_VP_HX_BDC    : BOOL;
    out_DO_VP_HX_HTR    : BOOL;
    out_DO_APT01        : BOOL;
    out_DO_APT02        : BOOL;
    out_DO_APT03        : BOOL;
    out_DO_APT04        : BOOL;
    out_DO_APT05        : BOOL;
    out_DO_P2           : BOOL;
    out_DO_P3           : BOOL;
    out_DO_P4           : BOOL;
    out_DO_PERS         : BOOL;
    out_P1_speed        : REAL;
    override_active     : BOOL;         (* TRUE si está sobreescribiendo *)
END_VAR

(* --- Implementación --- *)

override_active := test_active;

IF test_active THEN
    out_DO_V3V1         := tst_V3V1_B;
    out_DO_V3V2         := tst_V3V2_B;
    out_DO_V3V3         := tst_V3V3_B;
    out_DO_V3VSOL       := tst_V3VSOL_B;
    out_DO_VP_HX1       := tst_VP_HX1_open;
    out_DO_VP_HX_BDC    := tst_VP_HX_BDC_open;
    out_DO_VP_HX_HTR    := tst_VP_HX_HTR_open;
    out_DO_APT01        := tst_APT01_AFS;
    out_DO_APT02        := tst_APT02_AFS;
    out_DO_APT03        := tst_APT03_AFS;
    out_DO_APT04        := tst_APT04_AFS;
    out_DO_APT05        := tst_APT05_AFS;
    out_DO_P2           := tst_P2_on;
    out_DO_P3           := tst_P3_on;
    out_DO_P4           := tst_P4_on;
    out_DO_PERS         := tst_PERS_close;
    out_P1_speed        := LIMIT(0.0, tst_P1_speed_pct, 100.0);
ELSE
    (* Modo normal: no sobreescribir nada *)
    out_DO_V3V1         := FALSE;
    out_DO_V3V2         := FALSE;
    out_DO_V3V3         := FALSE;
    out_DO_V3VSOL       := FALSE;
    out_DO_VP_HX1       := FALSE;
    out_DO_VP_HX_BDC    := FALSE;
    out_DO_VP_HX_HTR    := FALSE;
    out_DO_APT01        := FALSE;
    out_DO_APT02        := FALSE;
    out_DO_APT03        := FALSE;
    out_DO_APT04        := FALSE;
    out_DO_APT05        := FALSE;
    out_DO_P2           := FALSE;
    out_DO_P3           := FALSE;
    out_DO_P4           := FALSE;
    out_DO_PERS         := FALSE;
    out_P1_speed        := 0.0;
END_IF

END_FUNCTION_BLOCK

(* ---- HMI_PRG.st ---- *)
(* ============================================================
   HMI_PRG.st
   Programa HMI del FREE Evolution.
   Display 4 dígitos 7-segmentos + teclas ▲▼ ENTER ESC F1 F2.

   ARQUITECTURA:
   - Usa library_SmartHMI de Eliwell (disponible en FREE Studio Plus)
   - Si SmartHMI no está disponible: sustituir FB_HMI_Page y
     FB_HMI_Item por los equivalentes del driver de display disponible.

   ESTRUCTURA DE MENÚS:
   [MAIN] → SOL / ACS / CLIM / PISC / APT / PAST / ALR / TEST / CFG

   CONVENCIONES DISPLAY 4 DÍGITOS:
   - Letras: abreviaturas 4 chars ("SOL." "ACS." "TT 1" "SP.5")
   - Números: con punto decimal cuando aplica ("27.0" "65.0")
   - Estados BOOL: " On " / " OFF"
   - Enums: "AUto" "PIsc" "AFS." "PREC"
   - Errores: "Err." "----" "HHH." "LLL."

   TECLAS:
   - ▲▼     Navegar entre ítems / cambiar valor
   - ENTER  Entrar en menú / confirmar edición
   - ESC    Volver al nivel superior / cancelar edición
   - F1     Acceso rápido a ALARMAS desde cualquier página
   - F2     Acceso rápido a página principal (MAIN)
   ============================================================ *)

PROGRAM HMI_PRG

VAR
    (* ---- Instancias SmartHMI (library_SmartHMI) ---- *)
    (* NOTA: Verificar nombres exactos de FB en FREE Studio Plus:
       Library Manager → library_SmartHMI → ver lista de FBs.
       Los nombres indicados aquí son los más probables según
       la documentación de la gama FREE. *)

    hmi             : FB_HMIController;     (* Controlador principal HMI *)

    (* Páginas principales *)
    pg_main         : FB_HMIPage;
    pg_sol          : FB_HMIPage;
    pg_acs          : FB_HMIPage;
    pg_clim         : FB_HMIPage;
    pg_pisc         : FB_HMIPage;
    pg_apt          : FB_HMIPage;
    pg_past         : FB_HMIPage;
    pg_alr          : FB_HMIPage;
    pg_test         : FB_HMIPage;
    pg_cfg          : FB_HMIPage;

    (* PIN guards *)
    pin_test        : FB_PIN_Guard;
    pin_cfg         : FB_PIN_Guard;
    pin_entered_val : UINT := 0;

    (* Test mode *)
    test_mode       : FB_TestMode;

    (* Auxiliares *)
    timer_alm_blink : TON;
    alm_blink_state : BOOL;
    any_alarm       : BOOL;

    (* Actividad panel (reset timeout sesión) *)
    panel_activity  : BOOL;

END_VAR

(* ============================================================
   1. GESTIÓN DE ALARMAS Y PARPADEO
   ============================================================ *)
any_alarm := alarms.CUALQUIER_ALARMA;

timer_alm_blink(IN := any_alarm, PT := T#500MS);
IF timer_alm_blink.Q THEN
    alm_blink_state := NOT alm_blink_state;
    timer_alm_blink(IN := FALSE, PT := T#500MS);
END_IF

(* ============================================================
   2. PROTECCIÓN PIN
   ============================================================ *)
pin_test(
    pin_stored      := HMI_pin_test,
    pin_entered     := pin_entered_val,
    confirm         := hmi.key_enter AND HMI_current_page = UINT#8,
    cancel          := hmi.key_esc,
    activity        := panel_activity,
    session_timeout := T#10M,
    lockout_time    := T#5M
);

pin_cfg(
    pin_stored      := HMI_pin_cfg,
    pin_entered     := pin_entered_val,
    confirm         := hmi.key_enter AND HMI_current_page = UINT#9,
    cancel          := hmi.key_esc,
    activity        := panel_activity,
    session_timeout := T#10M,
    lockout_time    := T#5M
);

HMI_test_active := pin_test.access_granted;
HMI_cfg_active  := pin_cfg.access_granted;

(* ============================================================
   3. MODO TEST
   ============================================================ *)
test_mode(test_active := HMI_test_active);
(* Las salidas de test_mode se aplican en PLC_PRG_Evolution *)

(* ============================================================
   4. DEFINICIÓN DE PÁGINAS HMI
   ============================================================
   NOTA IMPLEMENTACIÓN:
   En FREE Studio Plus con library_SmartHMI, cada FB_HMIPage
   se configura con:
     - title      : STRING (4 chars para 7-seg)
     - items[]    : array de FB_HMIItem
   Cada FB_HMIItem tiene:
     - label      : STRING (4 chars)
     - pVar       : POINTER TO variable
     - type       : READ_ONLY / EDITABLE / ACTION
     - min/max/step (para editables)
   La navegación es automática vía el FB_HMIController.
   ============================================================ *)

(* ---- PÁGINA MAIN ----------------------------------------- *)
(*
   Display muestra "MAIN"
   Items:
   [1] "SOL." → entrar pg_sol
   [2] "ACS." → entrar pg_acs
   [3] "CLIM" → entrar pg_clim
   [4] "PISC" → entrar pg_pisc
   [5] "APT." → entrar pg_apt
   [6] "PAST" → entrar pg_past
   [7] "ALR." → entrar pg_alr  ← parpadea si hay alarma activa
   [8] "TEST" → entrar pg_test (pide PIN)
   [9] "CFG." → entrar pg_cfg  (pide PIN)
*)
pg_main(
    title           := 'MAIN',
    show_alarm_icon := any_alarm
);

(* ---- PÁGINA SOLAR ---------------------------------------- *)
(*
   Label  | Variable              | Tipo        | Min  | Max   | Paso
   -------|----------------------|-------------|------|-------|------
   "TT 1" | SM.TT1               | READ_ONLY   |      |       |
   "TT 2" | TT2 (vía Modbus)     | READ_ONLY   |      |       |
   "TT 3" | SM.TT3               | READ_ONLY   |      |       |
   "d  T" | SM.DT_solar          | READ_ONLY   |      |       |
   "P  1" | SM.vel_P1 (→ % /10) | READ_ONLY   |      |       |
   "VLV." | SM.pos_V3V_SOL       | READ_ONLY   | ACS/PISC     |
   "PRS." | SM.persianas_cerr.   | READ_ONLY   | ABR/CER      |
   "SP.T" | HMI_SP_DT_solar      | EDITABLE    | 3.0  | 15.0  | 0.5
   "SP.P" | HMI_SP_TT3_pool      | EDITABLE    | 60.0 | 90.0  | 1.0
   "MOD." | HMI_modo_solar       | EDITABLE    | AUTO/ACS/PISC/OFF
*)
pg_sol(
    title           := 'SOL.',
    item_01_label   := 'TT 1', item_01_var := ADR(SM.TT1),           item_01_type := HMI_READ_ONLY,
    item_02_label   := 'TT 2', item_02_var := ADR(SM.TT2),           item_02_type := HMI_READ_ONLY,
    item_03_label   := 'TT 3', item_03_var := ADR(SM.TT3),           item_03_type := HMI_READ_ONLY,
    item_04_label   := 'd  T', item_04_var := ADR(SM.DT_solar),      item_04_type := HMI_READ_ONLY,
    item_05_label   := 'P  1', item_05_var := ADR(SM.vel_P1),        item_05_type := HMI_READ_ONLY,
    item_06_label   := 'SP.T', item_06_var := ADR(HMI_SP_DT_solar),  item_06_type := HMI_EDITABLE,
        item_06_min := 3.0,   item_06_max := 15.0,  item_06_step := 0.5,
    item_07_label   := 'SP.P', item_07_var := ADR(HMI_SP_TT3_pool),  item_07_type := HMI_EDITABLE,
        item_07_min := 60.0,  item_07_max := 90.0,  item_07_step := 1.0,
    item_08_label   := 'MOD.', item_08_var := ADR(HMI_modo_solar),   item_08_type := HMI_EDITABLE,
        item_08_min := 0,     item_08_max := 3,     item_08_step := 1
);

(* ---- PÁGINA ACS ------------------------------------------ *)
(*
   "TT 4" | TT4               | READ_ONLY
   "TT 5" | TT5               | READ_ONLY
   "SP.5" | HMI_SP_TT5        | EDITABLE  50-80  paso 0.5
   "HS.5" | HMI_HS_TT5        | EDITABLE  1.0-5.0 paso 0.5
   "SP.4" | HMI_SP_TT4_start  | EDITABLE  40-60  paso 0.5
   "V3.1" | DO_V3V1           | READ_ONLY (ACS/nAC)
   "V3.2" | DO_V3V2           | READ_ONLY (D3/HX)
   "V3.3" | DO_V3V3           | READ_ONLY (ACS/HX)
*)
pg_acs(
    title           := 'ACS.',
    item_01_label   := 'TT 4', item_01_var := ADR(TT4),              item_01_type := HMI_READ_ONLY,
    item_02_label   := 'TT 5', item_02_var := ADR(TT5),              item_02_type := HMI_READ_ONLY,
    item_03_label   := 'SP.5', item_03_var := ADR(HMI_SP_TT5),       item_03_type := HMI_EDITABLE,
        item_03_min := 50.0,  item_03_max := 80.0,  item_03_step := 0.5,
    item_04_label   := 'HS.5', item_04_var := ADR(HMI_HS_TT5),       item_04_type := HMI_EDITABLE,
        item_04_min := 1.0,   item_04_max := 5.0,   item_04_step := 0.5,
    item_05_label   := 'SP.4', item_05_var := ADR(HMI_SP_TT4_start), item_05_type := HMI_EDITABLE,
        item_05_min := 40.0,  item_05_max := 60.0,  item_05_step := 0.5,
    item_06_label   := 'V3.1', item_06_var := ADR(DO_V3V1),          item_06_type := HMI_READ_ONLY,
    item_07_label   := 'V3.2', item_07_var := ADR(DO_V3V2),          item_07_type := HMI_READ_ONLY,
    item_08_label   := 'V3.3', item_08_var := ADR(DO_V3V3),          item_08_type := HMI_READ_ONLY
);

(* ---- PÁGINA CLIMATIZACIÓN -------------------------------- *)
pg_clim(
    title           := 'CLIM',
    item_01_label   := 'TT 6', item_01_var := ADR(TT6),         item_01_type := HMI_READ_ONLY,
    item_02_label   := 'TT 7', item_02_var := ADR(TT7),         item_02_type := HMI_READ_ONLY,
    item_03_label   := 'SP.H', item_03_var := ADR(HMI_SP_heat), item_03_type := HMI_EDITABLE,
        item_03_min := 35.0,  item_03_max := 60.0, item_03_step := 0.5,
    item_04_label   := 'SP.C', item_04_var := ADR(HMI_SP_cool), item_04_type := HMI_EDITABLE,
        item_04_min := 5.0,   item_04_max := 15.0, item_04_step := 0.5,
    item_05_label   := 'HS.H', item_05_var := ADR(HMI_HS_heat), item_05_type := HMI_EDITABLE,
        item_05_min := 1.0,   item_05_max := 5.0,  item_05_step := 0.5,
    item_06_label   := 'HS.C', item_06_var := ADR(HMI_HS_cool), item_06_type := HMI_EDITABLE,
        item_06_min := 0.5,   item_06_max := 3.0,  item_06_step := 0.5,
    item_07_label   := 'P  3', item_07_var := ADR(DO_P3),       item_07_type := HMI_READ_ONLY
);

(* ---- PÁGINA PISCINA ------------------------------------- *)
pg_pisc(
    title           := 'PISC',
    item_01_label   := 'TT11', item_01_var := ADR(TT11),          item_01_type := HMI_READ_ONLY,
    item_02_label   := 'TT14', item_02_var := ADR(TT14),          item_02_type := HMI_READ_ONLY,
    item_03_label   := 'SP.P', item_03_var := ADR(HMI_SP_pool),   item_03_type := HMI_EDITABLE,
        item_03_min := 20.0,  item_03_max := 35.0, item_03_step := 0.5,
    item_04_label   := 'HS.P', item_04_var := ADR(HMI_HS_pool),   item_04_type := HMI_EDITABLE,
        item_04_min := 0.5,   item_04_max := 3.0,  item_04_step := 0.5,
    item_05_label   := 'VP.1', item_05_var := ADR(DO_VP_HX1),     item_05_type := HMI_READ_ONLY,
    item_06_label   := 'VP.B', item_06_var := ADR(DO_VP_HX_BDC),  item_06_type := HMI_READ_ONLY,
    item_07_label   := 'VP.H', item_07_var := ADR(DO_VP_HX_HTR),  item_07_type := HMI_READ_ONLY,
    item_08_label   := 'FLW.', item_08_var := ADR(DI_IF_PISC),    item_08_type := HMI_READ_ONLY
);

(* ---- PÁGINA APARTAMENTOS -------------------------------- *)
(*  Cada ítem: label "A 01"  valor: 0=PREC 1=AFS  *)
pg_apt(
    title           := 'APT.',
    item_01_label   := 'A 01', item_01_var := ADR(HMI_apt_mode_01), item_01_type := HMI_EDITABLE,
        item_01_min := 0, item_01_max := 1, item_01_step := 1,
    item_02_label   := 'A 02', item_02_var := ADR(HMI_apt_mode_02), item_02_type := HMI_EDITABLE,
        item_02_min := 0, item_02_max := 1, item_02_step := 1,
    item_03_label   := 'A 03', item_03_var := ADR(HMI_apt_mode_03), item_03_type := HMI_EDITABLE,
        item_03_min := 0, item_03_max := 1, item_03_step := 1,
    item_04_label   := 'A 04', item_04_var := ADR(HMI_apt_mode_04), item_04_type := HMI_EDITABLE,
        item_04_min := 0, item_04_max := 1, item_04_step := 1,
    item_05_label   := 'A 05', item_05_var := ADR(HMI_apt_mode_05), item_05_type := HMI_EDITABLE,
        item_05_min := 0, item_05_max := 1, item_05_step := 1
);

(* ---- PÁGINA PASTEURIZACIÓN ------------------------------ *)
pg_past(
    title           := 'PAST',
    item_01_label   := 'STA.', item_01_var := ADR(past_phase),        item_01_type := HMI_READ_ONLY,
    item_02_label   := 'TT 5', item_02_var := ADR(TT5),               item_02_type := HMI_READ_ONLY,
    item_03_label   := 'APT.', item_03_var := ADR(past_apt_idx),      item_03_type := HMI_READ_ONLY,
    item_04_label   := 'SP.T', item_04_var := ADR(HMI_SP_past_target),item_04_type := HMI_EDITABLE,
        item_04_min := 65.0,  item_04_max := 75.0, item_04_step := 0.5,
    item_05_label   := 'T.Ho', item_05_var := ADR(HMI_past_hold_min), item_05_type := HMI_EDITABLE,
        item_05_min := 30,    item_05_max := 120,  item_05_step := 5,
    item_06_label   := 'T.Fl', item_06_var := ADR(HMI_past_flush_min),item_06_type := HMI_EDITABLE,
        item_06_min := 15,    item_06_max := 60,   item_06_step := 5,
    item_07_label   := 'RUN.', item_07_var := ADR(HMI_req_past_manual),item_07_type := HMI_ACTION
);

(* ---- PÁGINA ALARMAS ------------------------------------- *)
(*  Cada alarma: label 4 chars, valor BOOL READ_ONLY
    "ACT." muestra el número de alarmas activas
    "RST." reset con ENTER                               *)
pg_alr(
    title           := 'ALR.',
    item_01_label   := 'ACT.', item_01_var := ADR(alm_count),             item_01_type := HMI_READ_ONLY,
    item_02_label   := 'TT1H', item_02_var := ADR(alarms.ALM_TT1_HIGH),   item_02_type := HMI_READ_ONLY,
    item_03_label   := 'TT2H', item_03_var := ADR(alarms.ALM_TT2_HIGH),   item_03_type := HMI_READ_ONLY,
    item_04_label   := 'COMM', item_04_var := ADR(alarms.ALM_COMM_SMART),  item_04_type := HMI_READ_ONLY,
    item_05_label   := 'TT5L', item_05_var := ADR(alarms.ALM_TT5_LOW),    item_05_type := HMI_READ_ONLY,
    item_06_label   := 'TT5H', item_06_var := ADR(alarms.ALM_TT5_HIGH),   item_06_type := HMI_READ_ONLY,
    item_07_label   := 'PFLW', item_07_var := ADR(alarms.ALM_PISC_FLUJO), item_07_type := HMI_READ_ONLY,
    item_08_label   := 'PTHH', item_08_var := ADR(alarms.ALM_PISC_T_HIGH),item_08_type := HMI_READ_ONLY,
    item_09_label   := 'INF.', item_09_var := ADR(alarms.ALM_INUNDACION),  item_09_type := HMI_READ_ONLY,
    item_10_label   := 'BDC.', item_10_var := ADR(alarms.ALM_BDC_FAULT),  item_10_type := HMI_READ_ONLY,
    item_11_label   := 'RST.', item_11_var := ADR(HMI_req_alm_reset),     item_11_type := HMI_ACTION
);

(* ---- PÁGINA TEST (requiere PIN) ------------------------- *)
pg_test(
    title           := 'TEST',
    locked          := NOT HMI_test_active,
    item_01_label   := 'P  1', item_01_var := ADR(test_mode.tst_P1_on),        item_01_type := HMI_EDITABLE,
        item_01_min := 0, item_01_max := 1, item_01_step := 1,
    item_02_label   := 'P1 %', item_02_var := ADR(test_mode.tst_P1_speed_pct), item_02_type := HMI_EDITABLE,
        item_02_min := 0.0, item_02_max := 100.0, item_02_step := 5.0,
    item_03_label   := 'P  2', item_03_var := ADR(test_mode.tst_P2_on),        item_03_type := HMI_EDITABLE,
        item_03_min := 0, item_03_max := 1, item_03_step := 1,
    item_04_label   := 'P  3', item_04_var := ADR(test_mode.tst_P3_on),        item_04_type := HMI_EDITABLE,
        item_04_min := 0, item_04_max := 1, item_04_step := 1,
    item_05_label   := 'P  4', item_05_var := ADR(test_mode.tst_P4_on),        item_05_type := HMI_EDITABLE,
        item_05_min := 0, item_05_max := 1, item_05_step := 1,
    item_06_label   := 'V3.1', item_06_var := ADR(test_mode.tst_V3V1_B),       item_06_type := HMI_EDITABLE,
        item_06_min := 0, item_06_max := 1, item_06_step := 1,
    item_07_label   := 'V3.2', item_07_var := ADR(test_mode.tst_V3V2_B),       item_07_type := HMI_EDITABLE,
        item_07_min := 0, item_07_max := 1, item_07_step := 1,
    item_08_label   := 'V3.3', item_08_var := ADR(test_mode.tst_V3V3_B),       item_08_type := HMI_EDITABLE,
        item_08_min := 0, item_08_max := 1, item_08_step := 1,
    item_09_label   := 'V3.S', item_09_var := ADR(test_mode.tst_V3VSOL_B),     item_09_type := HMI_EDITABLE,
        item_09_min := 0, item_09_max := 1, item_09_step := 1,
    item_10_label   := 'VP.1', item_10_var := ADR(test_mode.tst_VP_HX1_open),  item_10_type := HMI_EDITABLE,
        item_10_min := 0, item_10_max := 1, item_10_step := 1,
    item_11_label   := 'VP.B', item_11_var := ADR(test_mode.tst_VP_HX_BDC_open),item_11_type := HMI_EDITABLE,
        item_11_min := 0, item_11_max := 1, item_11_step := 1,
    item_12_label   := 'VP.H', item_12_var := ADR(test_mode.tst_VP_HX_HTR_open),item_12_type := HMI_EDITABLE,
        item_12_min := 0, item_12_max := 1, item_12_step := 1,
    item_13_label   := 'TA01', item_13_var := ADR(test_mode.tst_APT01_AFS),    item_13_type := HMI_EDITABLE,
        item_13_min := 0, item_13_max := 1, item_13_step := 1,
    item_14_label   := 'TA02', item_14_var := ADR(test_mode.tst_APT02_AFS),    item_14_type := HMI_EDITABLE,
        item_14_min := 0, item_14_max := 1, item_14_step := 1,
    item_15_label   := 'TA03', item_15_var := ADR(test_mode.tst_APT03_AFS),    item_15_type := HMI_EDITABLE,
        item_15_min := 0, item_15_max := 1, item_15_step := 1,
    item_16_label   := 'TA04', item_16_var := ADR(test_mode.tst_APT04_AFS),    item_16_type := HMI_EDITABLE,
        item_16_min := 0, item_16_max := 1, item_16_step := 1,
    item_17_label   := 'TA05', item_17_var := ADR(test_mode.tst_APT05_AFS),    item_17_type := HMI_EDITABLE,
        item_17_min := 0, item_17_max := 1, item_17_step := 1,
    item_18_label   := 'PRS.', item_18_var := ADR(test_mode.tst_PERS_close),   item_18_type := HMI_EDITABLE,
        item_18_min := 0, item_18_max := 1, item_18_step := 1,
    item_19_label   := 'EXT.', item_19_var := ADR(HMI_test_active),            item_19_type := HMI_ACTION
);

(* ---- PÁGINA CONFIGURACIÓN (requiere PIN) --------------- *)
pg_cfg(
    title           := 'CFG.',
    locked          := NOT HMI_cfg_active,
    item_01_label   := 'PRI.', item_01_var := ADR(HMI_bdc_priority),   item_01_type := HMI_EDITABLE,
        item_01_min := 0, item_01_max := 1, item_01_step := 1,
    item_02_label   := 'BDA.', item_02_var := ADR(HMI_mb_slave_addr),  item_02_type := HMI_EDITABLE,
        item_02_min := 1, item_02_max := 247, item_02_step := 1,
    item_03_label   := 'BDB.', item_03_var := ADR(HMI_mb_baudrate),    item_03_type := HMI_EDITABLE,
        item_03_min := 0, item_03_max := 2, item_03_step := 1,
    item_04_label   := 'PIN.', item_04_var := ADR(HMI_pin_test),       item_04_type := HMI_EDITABLE,
        item_04_min := 0, item_04_max := 9999, item_04_step := 1,
    item_05_label   := 'PIC.', item_05_var := ADR(HMI_pin_cfg),        item_05_type := HMI_EDITABLE,
        item_05_min := 0, item_05_max := 9999, item_05_step := 1,
    item_06_label   := 'RST.', item_06_var := ADR(HMI_req_factory_rst),item_06_type := HMI_ACTION
);

(* ============================================================
   5. CONTROLADOR HMI PRINCIPAL
   Conecta todas las páginas y gestiona la navegación.
   ============================================================ *)
hmi(
    pages           := [pg_main, pg_sol, pg_acs, pg_clim,
                        pg_pisc, pg_apt, pg_past, pg_alr,
                        pg_test, pg_cfg],
    root_page       := ADR(pg_main),
    alarm_blink     := alm_blink_state,
    key_f1_page     := ADR(pg_alr),     (* F1 → acceso directo alarmas *)
    key_f2_page     := ADR(pg_main)     (* F2 → volver al inicio *)
);

HMI_current_page := hmi.current_page_idx;
panel_activity   := hmi.any_key_pressed;

(* ============================================================
   6. PROPAGACIÓN DE SETPOINTS HMI → LÓGICA DE CONTROL
   Los setpoints editados en el panel se reflejan automáticamente
   en las constantes usadas por los FBs de control porque
   apuntan a las mismas variables GVL_HMI_Params (por referencia).
   No es necesario copiar valores — DRY: una sola variable.
   ============================================================ *)

(* Actualizar Modbus hacia FREE Smart con los setpoints editados *)
MB_TO_SMART_SP_DT       := REAL_TO_UINT(HMI_SP_DT_solar * MB_TEMP_SCALE);
MB_TO_SMART_MODO        := HMI_modo_solar;
MB_TO_SMART_SP_TT3_POOL := REAL_TO_UINT(HMI_SP_TT3_pool * MB_TEMP_SCALE);

END_PROGRAM

(* ---- PLC_PRG_Evolution.st ---- *)
(* ============================================================
   PLC_PRG_Evolution.st  –  Programa principal controlador principal
   Arquitectura: BC monobloc genérica (sin HTR) + solar térmico
   Task cíclica: 1000 ms
   Orden de ejecución:
     1. Aplicar offsets de sondas
     2. Polling Modbus controlador solar
     3. Higienización (máxima prioridad)
     4. Árbitro BDC
     5. ACS
     6. Climatización
     7. Piscina
     8. Apartamentos
     9. Modo test (sobreescribe salidas si activo)
    10. Escribir salidas físicas
    11. Alarmas
   ============================================================ *)
PROGRAM PLC_PRG

VAR
    (* ── Instancias de subsistemas ── *)
    mb_master       : FB_ModbusMaster;
    acs_ctrl        : FB_ACS;
    climate_ctrl    : FB_Climate;
    pool_ctrl       : FB_Pool;
    apt_ctrl        : FB_Apartments;
    bdc_arbiter     : FB_BDC_Arbiter;
    hyg_ctrl        : FB_Hygienization;
    alarms_ctrl     : FB_Alarms;
    test_ctrl       : FB_TestMode;

    (* ── Valores de sondas corregidos con offset ── *)
    TT4c  : REAL;  TT5c  : REAL;  TT6c  : REAL;  TT7c  : REAL;
    TT8c  : REAL;  TT9c  : REAL;  TT11c : REAL;
    TT12c : REAL;  TT13c : REAL;

    (* ── Auxiliares ── *)
    any_VP_open     : BOOL;
    alm_count_local : UINT;
    bdc_grant_pool  : BOOL;  (* BC a piscina solo si en modo calor *)
END_VAR

(* ============================================================
   1. APLICAR OFFSETS DE SONDAS
   ============================================================ *)
TT4c  := TT4  + OS03_TT4;
TT5c  := TT5  + OS04_TT5;
TT6c  := TT6  + OS05_TT6;
TT7c  := TT7  + OS06_TT7;
TT8c  := TT8  + OS07_TT8;
TT9c  := TT9  + OS08_TT9;
TT11c := TT11 + OS00_TT11;
TT12c := TT12 + OS00_TT12;
TT13c := TT13 + OS00_TT13;

(* ============================================================
   2. POLLING MODBUS  →  datos del controlador solar
   ============================================================ *)
mb_master(
    sp_dt_target    := P10_SolarDeltaTTarget,
    sp_tt3_pool     := P16_MinTempForPoolSolarHeating,
    sp_shutterclose := P17_SolarOverheatShutterClose,
    solar_mode      := P19_SolarMode,
    pool_demand     := pool_ctrl.demand_solar
);
SM := mb_master.solar;

(* ============================================================
   3. HIGIENIZACIÓN  (prioridad sobre todo)
   ============================================================ *)
hyg_ctrl(
    TT5            := TT5c,
    manual_request := hyg_request,
    enabled        := TRUE
);
hyg_phase   := hyg_ctrl.phase;
hyg_apt_idx := hyg_ctrl.apt_idx;

(* ============================================================
   4. ÁRBITRO BC
   ============================================================ *)
bdc_arbiter(
    demand_ACS     := acs_ctrl.demand_BDC OR hyg_ctrl.force_BDC_ACS,
    demand_climate := climate_ctrl.demand_BDC,
    demand_pool    := pool_ctrl.demand_BDC,
    enabled        := NOT DI_BDC_FAULT
);

(* La BC solo puede calentar la piscina en modo calor.
   En modo refrigeración su agua técnica está a 7-12°C. *)
bdc_grant_pool := bdc_arbiter.grant_pool AND bc_mode_heat;

(* ============================================================
   5. ACS
   ============================================================ *)
acs_ctrl(
    TT4           := TT4c,
    TT5           := TT5c,
    bdc_available := bdc_arbiter.grant_ACS,
    hyg_active    := hyg_ctrl.active,
    enabled       := TRUE
);

(* ============================================================
   6. CLIMATIZACIÓN
   ============================================================ *)
climate_ctrl(
    TT6           := TT6c,
    TT7           := TT7c,
    bdc_available := bdc_arbiter.grant_climate,
    mode_heat     := bc_mode_heat,
    enabled       := TRUE
);

(* ============================================================
   7. PISCINA
   ============================================================ *)
any_VP_open := DO_VP_HX_SOLAR OR DO_VP_HX_BC;
pool_ctrl(
    TT11           := TT11c,
    solar_available := SM.pos_V3V_SOL AND SM.P2_activo,
    bdc_available  := bdc_grant_pool,
    flow_ok        := DI_IF_PISC,
    enabled        := TRUE
);

(* ============================================================
   8. APARTAMENTOS
   ============================================================ *)
apt_ctrl(
    hyg_active       := hyg_ctrl.active,
    maintenance_mode := FALSE,
    enabled          := TRUE
);

(* ============================================================
   9. MODO TEST  (sobreescribe salidas si activo)
   ============================================================ *)
test_ctrl(test_active := HMI_test_active);

(* ============================================================
   10. ESCRIBIR SALIDAS DIGITALES
   ============================================================ *)
IF test_ctrl.override_active THEN
    DO_V3V1        := test_ctrl.out_DO_V3V1;
    DO_V3V2        := test_ctrl.out_DO_V3V2;
    DO_VP_HX_SOLAR := test_ctrl.out_DO_VP_HX1;
    DO_VP_HX_BC    := test_ctrl.out_DO_VP_HX_BDC;
    DO_V3V_APT_01  := test_ctrl.out_DO_APT01;
    DO_V3V_APT_02  := test_ctrl.out_DO_APT02;
    DO_V3V_APT_03  := test_ctrl.out_DO_APT03;
    DO_V3V_APT_04  := test_ctrl.out_DO_APT04;
    DO_P3          := test_ctrl.out_DO_P3;
ELSE
    (* Salidas normales *)
    (* V3V1: FALSE=reservorio (D2), TRUE=→V3V2 *)
    DO_V3V1        := NOT acs_ctrl.cmd_V3V1_reservorio AND NOT hyg_ctrl.force_BDC_ACS;
    (* V3V2: FALSE=fancoils (D3), TRUE=piscina (HX_BC) *)
    DO_V3V2        := pool_ctrl.cmd_VP_HX_BC AND NOT climate_ctrl.cmd_V3V2_D3;
    DO_VP_HX_SOLAR := pool_ctrl.cmd_VP_HX_SOLAR;
    DO_VP_HX_BC    := pool_ctrl.cmd_VP_HX_BC;
    DO_V3V_APT_01  := apt_ctrl.cmd_APT_01;
    DO_V3V_APT_02  := apt_ctrl.cmd_APT_02;
    DO_V3V_APT_03  := apt_ctrl.cmd_APT_03;
    DO_V3V_APT_04  := apt_ctrl.cmd_APT_04;
    DO_P3          := climate_ctrl.cmd_P3;
END_IF

(* ============================================================
   11. ALARMAS
   ============================================================ *)
alarms_ctrl(
    TT1           := SM.TT1,
    TT2           := SM.TT2,
    TT5           := TT5c,
    TT11          := TT11c,
    comm_solar_ok := SM.comm_ok,
    flow_pisc_ok  := DI_IF_PISC,
    vp_any_open   := any_VP_open,
    inundacion    := DI_INUND_FC,
    bdc_fault     := DI_BDC_FAULT,
    reset_cmd     := HMI_req_alm_reset,
    enabled       := TRUE
);
alarms          := alarms_ctrl.alarms;
alm_count_local := alarms_ctrl.alarm_count;

IF HMI_req_alm_reset THEN
    HMI_req_alm_reset := FALSE;
END_IF

END_PROGRAM
